# B&R Automation Studio project Lecture_10_jbl
Automation Studio 4.8.2.72

## Configuration Config1

### Task classes (Cpu.sw)
```
Cyclic#4:
  Assignment <- Assignment1.prg
  Assignmen1 <- Assignment2.prg
Libraries: AsTCP, runtime, AsBrStr
```

## Logical view

### Program Logical/Assignment1

#### Main.st
```iecst
PROGRAM _INIT
	tcpst := TCPSTATE_SOCKET_OPEN;

END_PROGRAM

PROGRAM _CYCLIC
	CASE tcpst OF
		TCPSTATE_SOCKET_OPEN :
			TcpOpen1.enable := TRUE;
			TcpOpen1.port := 12345;
			TcpOpen1.options := tcpOPT_REUSEADDR;
			TcpOpen1();
			IF (TcpOpen1.status = ERR_OK) THEN
				tcpst := TCPSTATE_SERVER_CREATE;
			END_IF

		TCPSTATE_SERVER_CREATE :
			TcpServer1.enable := TRUE;
			TcpServer1.ident := TcpOpen1.ident;
			TcpServer1();
			IF (TcpServer1.status = ERR_OK) THEN
				tcpst := TCPSTATE_RECEIVE;
			END_IF

		TCPSTATE_RECEIVE :
			TcpReceive1.enable := TRUE;
			TcpReceive1.ident := TcpServer1.identclnt;
			TcpReceive1.pData := ADR(receiveData);
			TcpReceive1.datamax := SIZEOF(receiveData);
			TcpReceive1();
			IF (TcpReceive1.status = ERR_OK) THEN
				tcpst := TCPSTATE_SEND;
				sendData := receiveData;
			END_IF

		TCPSTATE_SEND :
			TcpSend1.enable := TRUE;
			TcpSend1.ident := TcpServer1.identclnt;
			TcpSend1.pData := ADR(sendData);
			TcpSend1.datalen := brsstrlen(ADR(sendData));     // We use brsstrlen() to get the length in UDINT datatype
			TcpSend1();
			IF (TcpSend1.status = ERR_OK) THEN
				tcpst := TCPSTATE_CLOSE;
			END_IF

		TCPSTATE_CLOSE :
			TcpClose1.enable := TRUE;
			TcpClose1.ident := TcpServer1.identclnt;
			TcpClose1();
			IF (TcpClose1.status = ERR_OK) THEN
				TcpServer1.enable := FALSE;
				TcpServer1();
				tcpst := TCPSTATE_SERVER_CREATE;
			END_IF

	END_CASE

END_PROGRAM

PROGRAM _EXIT
	TcpClose1.enable := TRUE;
	TcpClose1.ident := TcpServer1.identclnt;
	TcpClose1();

	TcpClose2.enable := TRUE;
	TcpClose2.ident := TcpOpen1.ident;
	TcpClose2();

END_PROGRAM
```

### Program Logical/Assignment2

#### Variables.var
```iecst
VAR
	data1 : STRING[80];
	data2 : STRING[80];
	tcpst : TCPSTATE;
	sendData : STRING[80];
	receiveData : STRING[80];
	TcpOpen1 : TcpOpen;
	TcpServer1 : TcpServer;
	TcpReceive1 : TcpRecv;
	TcpSend1 : TcpSend;
	TcpClose1 : TcpClose;
	TcpClose2 : TcpClose;
	testUA : INT;
END_VAR
```

#### Main.st
```iecst
PROGRAM _INIT
	tcpst := TCPSTATE_SOCKET_OPEN;

END_PROGRAM

PROGRAM _CYCLIC
	CASE tcpst OF
		TCPSTATE_SOCKET_OPEN :
			TcpOpen1.enable := TRUE;
			TcpOpen1.port := 12345;
			TcpOpen1.options := tcpOPT_REUSEADDR;
			TcpOpen1();
			IF (TcpOpen1.status = ERR_OK) THEN
				tcpst := TCPSTATE_SERVER_CREATE;
			END_IF

		TCPSTATE_SERVER_CREATE :
			TcpServer1.enable := TRUE;
			TcpServer1.ident := TcpOpen1.ident;
			TcpServer1();
			IF (TcpServer1.status = ERR_OK) THEN
				tcpst := TCPSTATE_RECEIVE;
			END_IF

		TCPSTATE_RECEIVE :
			TcpReceive1.enable := TRUE;
			TcpReceive1.ident := TcpServer1.identclnt;
			TcpReceive1.pData := ADR(receiveData);
			TcpReceive1.datamax := SIZEOF(receiveData);
			TcpReceive1();
			IF (TcpReceive1.status = ERR_OK) THEN
				tcpst := TCPSTATE_SEND;
				sendData := receiveData;
				IF processReady AND SIZEOF(data1) := 0;
					data1 := receiveData;
				ELSE
					data2 := receiveData;
				END_IF
			END_IF

		TCPSTATE_SEND :
			TcpSend1.enable := TRUE;
			TcpSend1.ident := TcpServer1.identclnt;
			TcpSend1.pData := ADR(sendData);
			TcpSend1.datalen := brsstrlen(ADR(sendData));     // We use brsstrlen() to get the length in UDINT datatype
			TcpSend1();
			IF (TcpSend1.status = ERR_OK) THEN
				tcpst := TCPSTATE_CLOSE;
			END_IF

		TCPSTATE_CLOSE :
			TcpClose1.enable := TRUE;
			TcpClose1.ident := TcpServer1.identclnt;
			TcpClose1();
			IF (TcpClose1.status = ERR_OK) THEN
				TcpServer1.enable := FALSE;
				TcpServer1();
				tcpst := TCPSTATE_SERVER_CREATE;
			END_IF

	END_CASE

END_PROGRAM

PROGRAM _EXIT
	TcpClose1.enable := TRUE;
	TcpClose1.ident := TcpServer1.identclnt;
	TcpClose1();

	TcpClose2.enable := TRUE;
	TcpClose2.ident := TcpOpen1.ident;
	TcpClose2();

END_PROGRAM
```
